{attribute addProperty BoxType "EK1122-0000-0018"}
{attribute addProperty Id "Beckhoff_EPP7xxxsub_EK1100EK1100_179A0949162A_0001_EPP7041_1002_0016EPP7041_4CF4B42922628.25A_0002_EPP7041_1002_0017EPP7041_4CF4B42922628.25A_0003_EPP7041_1002_0023EPP7041_F30AD12822628.25A_0004_EPP7041_3002_0016EPP7041_F30AD12822628.25A_0005_EPP7041_3002_0017EPP7041_F30AD12822628.25A_0006_EPP7041_3002_0018EPP7041_F30AD12822628.25A_0007_EPP7041_3002_0023EPP7041_F30AD12822628.25A_0008_EPP7342_0002_0016EPP7342_E2585B8337046.25A_0009_EPP7342_0002_0017EPP7342_E2585B8337046.25"}
{attribute addProperty CRC "219269691"}
{attribute addProperty SizeInBites "2338"}
{attribute addProperty SizeInBytes "292.25"}
TYPE Beckhoff_EPP7xxxEK1122_0D11CA3B EXTENDS EK1122_179A0949 :
STRUCT
	{attribute addProperty Name "Beckhoff_EPP7xxxsub_EK1100"}
	Beckhoff_EPP7xxxsub_EK1100 : EK1100_179A0949;
	{attribute addProperty Name "A_0001_EPP7041_1002_0016"}
	A_0001_EPP7041_1002_0016 : EPP7041_4CF4B429;
	{attribute addProperty Name "A_0002_EPP7041_1002_0017"}
	A_0002_EPP7041_1002_0017 : EPP7041_4CF4B429;
	{attribute addProperty Name "A_0003_EPP7041_1002_0023"}
	A_0003_EPP7041_1002_0023 : EPP7041_F30AD128;
	{attribute addProperty Name "A_0004_EPP7041_3002_0016"}
	A_0004_EPP7041_3002_0016 : EPP7041_F30AD128;
	{attribute addProperty Name "A_0005_EPP7041_3002_0017"}
	A_0005_EPP7041_3002_0017 : EPP7041_F30AD128;
	{attribute addProperty Name "A_0006_EPP7041_3002_0018"}
	A_0006_EPP7041_3002_0018 : EPP7041_F30AD128;
	{attribute addProperty Name "A_0007_EPP7041_3002_0023"}
	A_0007_EPP7041_3002_0023 : EPP7041_F30AD128;
	{attribute addProperty Name "A_0008_EPP7342_0002_0016"}
	A_0008_EPP7342_0002_0016 : EPP7342_E2585B83;
	{attribute addProperty Name "A_0009_EPP7342_0002_0017"}
	A_0009_EPP7342_0002_0017 : EPP7342_E2585B83;
END_STRUCT
END_TYPE

(* stored: Version 1.2.0.0, ProductVersion 3.1.4024.9
   DUT Beckhoff_EPP7xxxEK1122_0D11CA3B: Id {de06763e-4d74-4208-a4c6-effa27833438} *)
